# B&R Automation Studio project MVP_ACOPOStrak (part 2)

#### Cyclic.st - Cyclic code
```iecst
PROGRAM _CYCLIC
	CASE Step OF
		CHECK_TRIGGER:
(* When the process is enabled and the assembly is ready,
the process will be activated *)
			IF((CmdEnableProcess) AND (gTrakAsm.Status.Ready))THEN
				MC_BR_TrgPointEnable_AcpTrak_0.Enable := TRUE;
(* If a shuttle passes the triggerpoint then
get the axis reference *)
				IF((MC_BR_TrgPointEnable_AcpTrak_0.Valid) AND
					(MC_BR_TrgPointEnable_AcpTrak_0.EventCount > 0))THEN
					MC_BR_TrgPointGetInfo_AcpTrak_0.Execute := TRUE;
				END_IF
			ELSE (* Else the processpoint will be disabled *)
				MC_BR_TrgPointEnable_AcpTrak_0.Enable := FALSE;
			END_IF
(* If axis reference is available,
save it AND go TO the next step *)
			IF EDGEPOS(MC_BR_TrgPointGetInfo_AcpTrak_0.Done) THEN
(* Save axis reference in local variable for use
in step machine *)
				ShuttleAxis := MC_BR_TrgPointGetInfo_AcpTrak_0.TrgPointInfo.Axis;
				MC_BR_TrgPointGetInfo_AcpTrak_0.Execute := FALSE;
				Step := GET_USERDATA;
				END_IF

		GET_USERDATA:
			(* The userdata is copied on a local variable *)
			MC_BR_ShCopyUserData_AcpTrak_0.Axis := ADR(ShuttleAxis);
			MC_BR_ShCopyUserData_AcpTrak_0.Execute := TRUE;
			MC_BR_ShCopyUserData_AcpTrak_0.DataAddress := ADR(ShuttleUserData);
			MC_BR_ShCopyUserData_AcpTrak_0.DataSize := SIZEOF(ShuttleUserData);
			MC_BR_ShCopyUserData_AcpTrak_0.Mode := mcACPTRAK_USERDATA_GET;
					(* After copying go to the next step *)

			IF EDGEPOS(MC_BR_ShCopyUserData_AcpTrak_0.Done) THEN
				MC_BR_ShCopyUserData_AcpTrak_0.Execute := FALSE;
				Step := PROCESS;
					END_IF

		PROCESS:

			CASE SubStep OF
				0:

					MC_BR_RoutedMoveAbs_AcpTrak_0.Axis := ADR(ShuttleAxis);
					MC_BR_BarrierCommand_AcpTrak_0.Execute := FALSE;

					IF ShuttleUserData.Task = PartsToCell1 OR ShuttleUserData.Task = PartsToCell2 OR ShuttleUserData.Task = MoveAssembly OR ShuttleUserData.Task = MoveSubAssembly THEN
						MC_BR_RoutedMoveAbs_AcpTrak_0.Execute := TRUE;
						MC_BR_RoutedMoveAbs_AcpTrak_0.Sector := ADR(SubSector1_1);
						MC_BR_RoutedMoveAbs_AcpTrak_0.Position := 0.68;
						MC_BR_RoutedMoveAbs_AcpTrak_0.Velocity := 2;
						MC_BR_RoutedMoveAbs_AcpTrak_0.Acceleration := 40;
						MC_BR_RoutedMoveAbs_AcpTrak_0.Deceleration := 40;
						MC_BR_RoutedMoveAbs_AcpTrak_0.Jerk := 0.0;
						MC_BR_RoutedMoveAbs_AcpTrak_0.AdvancedParameters.StartDirection := mcDIR_UNDEFINED;
						MC_BR_RoutedMoveAbs_AcpTrak_0.AdvancedParameters.ShuttleOrientation := mcDIR_POSITIVE;
						MC_BR_RoutedMoveAbs_AcpTrak_0.AdvancedParameters.EndDirection := mcDIR_UNDEFINED;

						IF EDGEPOS (MC_BR_RoutedMoveAbs_AcpTrak_0.Done) THEN
							MC_BR_RoutedMoveAbs_AcpTrak_0.Execute := FALSE;
							SubStep := 10;
						END_IF
					ELSE
						Step := SET_USERDATA;

					END_IF

				10:

					MC_BR_RoutedMoveAbs_AcpTrak_0.Axis := ADR(ShuttleAxis);
					MC_BR_RoutedMoveAbs_AcpTrak_0.Execute := TRUE;

					MC_BR_RoutedMoveAbs_AcpTrak_0.Sector := ADR(SectorTrack6);
					MC_BR_RoutedMoveAbs_AcpTrak_0.Position := 0.1;
					MC_BR_RoutedMoveAbs_AcpTrak_0.Velocity := 2;
					MC_BR_RoutedMoveAbs_AcpTrak_0.Acceleration := 40;
					MC_BR_RoutedMoveAbs_AcpTrak_0.Deceleration := 40;
					MC_BR_RoutedMoveAbs_AcpTrak_0.Jerk := 0.0;
					MC_BR_RoutedMoveAbs_AcpTrak_0.AdvancedParameters.StartDirection := mcDIR_UNDEFINED;
					MC_BR_RoutedMoveAbs_AcpTrak_0.AdvancedParameters.ShuttleOrientation := mcDIR_UNDEFINED;
					MC_BR_RoutedMoveAbs_AcpTrak_0.AdvancedParameters.EndDirection := mcDIR_UNDEFINED;

					IF EDGEPOS (MC_BR_RoutedMoveAbs_AcpTrak_0.Done) THEN
						WaitingLoadOn := TRUE;
					END_IF

					IF LoadOnTrack THEN
						MC_BR_RoutedMoveAbs_AcpTrak_0.Execute := FALSE;
						WaitingLoadOn := FALSE;
						LoadOnTrack := FALSE;
						MC_BR_BarrierCommand_AcpTrak_0.Execute := TRUE;
						MC_BR_BarrierCommand_AcpTrak_0.Command := 1;
						SubStep := 20;
					END_IF

				20:

					MC_BR_BarrierCommand_AcpTrak_0.Execute := FALSE;
					MC_BR_BarrierCommand_AcpTrak_0.Command := 0;
					MC_BR_RoutedMoveAbs_AcpTrak_0.Axis := ADR(ShuttleAxis);
					MC_BR_RoutedMoveAbs_AcpTrak_0.Execute := TRUE;

					MC_BR_RoutedMoveAbs_AcpTrak_0.Sector := ADR(SectorTrack1);
					MC_BR_RoutedMoveAbs_AcpTrak_0.Position := 13;
					MC_BR_RoutedMoveAbs_AcpTrak_0.Velocity := Speed_PP_04;
					MC_BR_RoutedMoveAbs_AcpTrak_0.Acceleration := 20;
					MC_BR_RoutedMoveAbs_AcpTrak_0.Deceleration := 20;
					MC_BR_RoutedMoveAbs_AcpTrak_0.Jerk := 0.0;
					MC_BR_RoutedMoveAbs_AcpTrak_0.AdvancedParameters.StartDirection := mcDIR_UNDEFINED;
					MC_BR_RoutedMoveAbs_AcpTrak_0.AdvancedParameters.ShuttleOrientation := mcDIR_POSITIVE;
					MC_BR_RoutedMoveAbs_AcpTrak_0.AdvancedParameters.EndDirection := mcDIR_UNDEFINED;

					IF EDGEPOS (MC_BR_RoutedMoveAbs_AcpTrak_0.Active) THEN
						MC_BR_RoutedMoveAbs_AcpTrak_0.Execute := FALSE;
						TON_0.IN := TRUE;
						TON_0.PT := T#2s;
						SubStep := 0;
						Step := SET_USERDATA;
					END_IF

			END_CASE

		SET_USERDATA:
			(* The modified userdata will be copied back on the shuttle *)
			MC_BR_ShCopyUserData_AcpTrak_0.Axis := ADR(ShuttleAxis);
			MC_BR_ShCopyUserData_AcpTrak_0.Execute := TRUE;
			MC_BR_ShCopyUserData_AcpTrak_0.DataAddress := ADR(ShuttleUserData);
			MC_BR_ShCopyUserData_AcpTrak_0.DataSize := SIZEOF(ShuttleUserData);
			MC_BR_ShCopyUserData_AcpTrak_0.Mode := mcACPTRAK_USERDATA_SET;

			(* After copying go to the first step and wait for new event *)
			IF EDGEPOS(MC_BR_ShCopyUserData_AcpTrak_0.Done) THEN
				MC_BR_ShCopyUserData_AcpTrak_0.Execute := FALSE;
				Step := CHECK_TRIGGER;
			END_IF
	END_CASE

	IF TON_0.Q THEN
		TON_0.IN := FALSE;
		Track6_Occupied := FALSE;
		MC_BR_BarrierCommand_AcpTrak_0.Execute := TRUE;
	END_IF

	(* Call all function blocks *)
	MC_BR_TrgPointEnable_AcpTrak_0();
	MC_BR_TrgPointGetInfo_AcpTrak_0();
	MC_BR_ShCopyUserData_AcpTrak_0();
	MC_BR_RoutedMoveAbs_AcpTrak_0();
	MC_BR_BarrierCommand_AcpTrak_0();
	TON_0();

END_PROGRAM
PROGRAM _EXIT
END_PROGRAM
```

#### Init.st - Init code
```iecst
PROGRAM _INIT
(* Local variable to enable/disable the the process *)
	Speed_PP_04 := 2;
	CmdEnableProcess := TRUE;
	(* Processpointreference for Functionblocks *)
	MC_BR_TrgPointEnable_AcpTrak_0.ProcessPoint := ADR(PP1);
	MC_BR_TrgPointGetInfo_AcpTrak_0.ProcessPoint := ADR(PP1);
END_PROGRAM
```

#### Types.typ - Local data types
```iecst
TYPE
	Step_enum :
		(
		CHECK_TRIGGER,
		GET_USERDATA,
		PROCESS,
		SET_USERDATA
	);
END_TYPE
```

#### Variables.var - Local variables
```iecst
VAR
	Speed_PP_04 : {REDUND_UNREPLICABLE} REAL := 0.0;
	MC_BR_BarrierCommand_AcpTrak_0 : MC_BR_BarrierCommand_AcpTrak;
	Step : Step_enum;
	MC_BR_TrgPointEnable_AcpTrak_0 : MC_BR_TrgPointEnable_AcpTrak;
	CmdEnableProcess : BOOL;
	MC_BR_TrgPointGetInfo_AcpTrak_0 : MC_BR_TrgPointGetInfo_AcpTrak;
	ShuttleAxis : McAxisType;
	MC_BR_ShCopyUserData_AcpTrak_0 : MC_BR_ShCopyUserData_AcpTrak;
	MC_BR_RoutedMoveAbs_AcpTrak_0 : MC_BR_RoutedMoveAbs_AcpTrak;
	SubStep : UDINT;
	TaskReady : BOOL;
	TON_0 : TON;
	ShuttleUserData : ShuttleUserData_typ;
	MC_BR_RoutedMoveVel_AcpTrak_0 : MC_BR_RoutedMoveVel_AcpTrak;
END_VAR
```

### Program Logical/PP2 (IEC)

#### Variables.var
```iecst
VAR
	Speed_PP_04 : {REDUND_UNREPLICABLE} REAL := 0.0;
	MC_BR_BarrierCommand_AcpTrak_0 : MC_BR_BarrierCommand_AcpTrak;
	Step : Step_enum;
	MC_BR_TrgPointEnable_AcpTrak_0 : MC_BR_TrgPointEnable_AcpTrak;
	CmdEnableProcess : BOOL;
	MC_BR_TrgPointGetInfo_AcpTrak_0 : MC_BR_TrgPointGetInfo_AcpTrak;
	ShuttleAxis : McAxisType;
	MC_BR_ShCopyUserData_AcpTrak_0 : MC_BR_ShCopyUserData_AcpTrak;
	MC_BR_RoutedMoveVel_AcpTrak_0 : MC_BR_RoutedMoveVel_AcpTrak;
	SubStep : UDINT;
	TaskReady : BOOL;
	TaskCompleteCell1 : BOOL;
	ShuttleUserData : ShuttleUserData_typ;
END_VAR
```

#### Cyclic.st
```iecst
PROGRAM _CYCLIC
	CASE Step OF
		CHECK_TRIGGER:
(* When the process is enabled and the assembly is ready,
the process will be activated *)
			IF((CmdEnableProcess) AND (gTrakAsm.Status.Ready))THEN
				MC_BR_TrgPointEnable_AcpTrak_0.Enable := TRUE;
(* If a shuttle passes the triggerpoint then
get the axis reference *)
				IF((MC_BR_TrgPointEnable_AcpTrak_0.Valid) AND
					(MC_BR_TrgPointEnable_AcpTrak_0.EventCount > 0))THEN
					MC_BR_TrgPointGetInfo_AcpTrak_0.Execute := TRUE;
				END_IF
			ELSE (* Else the processpoint will be disabled *)
				MC_BR_TrgPointEnable_AcpTrak_0.Enable := FALSE;
			END_IF
(* If axis reference is available,
save it AND go TO the next step *)
			IF EDGEPOS(MC_BR_TrgPointGetInfo_AcpTrak_0.Done) THEN
(* Save axis reference in local variable for use
in step machine *)
				ShuttleAxis := MC_BR_TrgPointGetInfo_AcpTrak_0.TrgPointInfo.Axis;
				MC_BR_TrgPointGetInfo_AcpTrak_0.Execute := FALSE;
				Step := GET_USERDATA;
				END_IF

		GET_USERDATA:
			(* The userdata is copied on a local variable *)
			MC_BR_ShCopyUserData_AcpTrak_0.Axis := ADR(ShuttleAxis);
			MC_BR_ShCopyUserData_AcpTrak_0.Execute := TRUE;
			MC_BR_ShCopyUserData_AcpTrak_0.DataAddress := ADR(ShuttleUserData);
			MC_BR_ShCopyUserData_AcpTrak_0.DataSize := SIZEOF(ShuttleUserData);
			MC_BR_ShCopyUserData_AcpTrak_0.Mode := mcACPTRAK_USERDATA_GET;
					(* After copying go to the next step *)

			IF EDGEPOS(MC_BR_ShCopyUserData_AcpTrak_0.Done) THEN
				MC_BR_ShCopyUserData_AcpTrak_0.Execute := FALSE;
				Step := PROCESS;
					END_IF

		PROCESS:

		IF ShuttleUserData.Task = PartsToCell1 OR ShuttleUserData.Task = PartsFromCell1 OR ShuttleUserData.Task = MoveAssembly THEN

			MC_BR_RoutedMoveVel_AcpTrak_0.Axis := ADR(ShuttleAxis);
			MC_BR_RoutedMoveVel_AcpTrak_0.Execute := TRUE;
			MC_BR_RoutedMoveVel_AcpTrak_0.Sector := ADR(SectorTrack2);
			MC_BR_RoutedMoveVel_AcpTrak_0.Position := 0;
			MC_BR_RoutedMoveVel_AcpTrak_0.Velocity := Speed_PP_04;
			MC_BR_RoutedMoveVel_AcpTrak_0.RouteVelocity := Speed_PP_04;
			MC_BR_RoutedMoveVel_AcpTrak_0.Acceleration := 10;
			MC_BR_RoutedMoveVel_AcpTrak_0.Deceleration := 10;
			MC_BR_RoutedMoveVel_AcpTrak_0.Jerk := 0.0;
			MC_BR_RoutedMoveVel_AcpTrak_0.AdvancedParameters.StartDirection := mcDIR_UNDEFINED;
			MC_BR_RoutedMoveVel_AcpTrak_0.AdvancedParameters.ShuttleOrientation := mcDIR_NEGATIVE;
			MC_BR_RoutedMoveVel_AcpTrak_0.AdvancedParameters.EndDirection := mcDIR_UNDEFINED;

			IF EDGEPOS (MC_BR_RoutedMoveVel_AcpTrak_0.Active) THEN
				MC_BR_RoutedMoveVel_AcpTrak_0.Execute := FALSE;
				Step := SET_USERDATA;
				END_IF
			ELSE

				MC_BR_RoutedMoveVel_AcpTrak_0.Axis := ADR(ShuttleAxis);
				MC_BR_RoutedMoveVel_AcpTrak_0.Execute := TRUE;
				MC_BR_RoutedMoveVel_AcpTrak_0.Sector := ADR(SectorTrack1);
				MC_BR_RoutedMoveVel_AcpTrak_0.Position := 5;
				MC_BR_RoutedMoveVel_AcpTrak_0.Velocity := Speed_PP_04;
				MC_BR_RoutedMoveVel_AcpTrak_0.RouteVelocity := Speed_PP_04;
				MC_BR_RoutedMoveVel_AcpTrak_0.Acceleration := 10;
				MC_BR_RoutedMoveVel_AcpTrak_0.Deceleration := 10;
				MC_BR_RoutedMoveVel_AcpTrak_0.Jerk := 0.0;
				MC_BR_RoutedMoveVel_AcpTrak_0.AdvancedParameters.StartDirection := mcDIR_POSITIVE;
				MC_BR_RoutedMoveVel_AcpTrak_0.AdvancedParameters.ShuttleOrientation := mcDIR_UNDEFINED;
				MC_BR_RoutedMoveVel_AcpTrak_0.AdvancedParameters.EndDirection := mcDIR_UNDEFINED;

				IF EDGEPOS (MC_BR_RoutedMoveVel_AcpTrak_0.Active) THEN
					MC_BR_RoutedMoveVel_AcpTrak_0.Execute := FALSE;
					Step := SET_USERDATA;
				END_IF
		END_IF

		SET_USERDATA:
			(* The modified userdata will be copied back on the shuttle *)
			MC_BR_ShCopyUserData_AcpTrak_0.Axis := ADR(ShuttleAxis);
			MC_BR_ShCopyUserData_AcpTrak_0.Execute := TRUE;
			MC_BR_ShCopyUserData_AcpTrak_0.DataAddress := ADR(ShuttleUserData);
			MC_BR_ShCopyUserData_AcpTrak_0.DataSize := SIZEOF(ShuttleUserData);
			MC_BR_ShCopyUserData_AcpTrak_0.Mode := mcACPTRAK_USERDATA_SET;

			(* After copying go to the first step and wait for new event *)
			IF EDGEPOS(MC_BR_ShCopyUserData_AcpTrak_0.Done) THEN
				MC_BR_ShCopyUserData_AcpTrak_0.Execute := FALSE;
				Step := CHECK_TRIGGER;
			END_IF
	END_CASE

	(* Call all function blocks *)
	MC_BR_TrgPointEnable_AcpTrak_0();
	MC_BR_TrgPointGetInfo_AcpTrak_0();
	MC_BR_ShCopyUserData_AcpTrak_0();
	MC_BR_RoutedMoveVel_AcpTrak_0();
	MC_BR_BarrierCommand_AcpTrak_0();

END_PROGRAM
PROGRAM _EXIT
END_PROGRAM
```

#### Init.st
```iecst
PROGRAM _INIT
(* Local variable to enable/disable the the process *)
	Speed_PP_04 := 2;
	CmdEnableProcess := TRUE;
	(* Processpointreference for Functionblocks *)
	MC_BR_TrgPointEnable_AcpTrak_0.ProcessPoint := ADR(PP2);
	MC_BR_TrgPointGetInfo_AcpTrak_0.ProcessPoint := ADR(PP2);
END_PROGRAM
```

### Program Logical/PB2 (IEC)

#### Variables.var
```iecst
VAR
	Speed_PP_04 : {REDUND_UNREPLICABLE} REAL := 0.0;
	MC_BR_BarrierCommand_AcpTrak_0 : MC_BR_BarrierCommand_AcpTrak;
	Step : Step_enum;
	MC_BR_TrgPointEnable_AcpTrak_0 : MC_BR_TrgPointEnable_AcpTrak;
	CmdEnableProcess : BOOL;
	MC_BR_TrgPointGetInfo_AcpTrak_0 : MC_BR_TrgPointGetInfo_AcpTrak;
	ShuttleAxis : McAxisType;
	MC_BR_ShCopyUserData_AcpTrak_0 : MC_BR_ShCopyUserData_AcpTrak;
	MC_BR_RoutedMoveAbs_AcpTrak_0 : MC_BR_RoutedMoveAbs_AcpTrak;
	SubStep : UDINT;
	TaskReady : BOOL;
	MC_BR_RoutedMoveVel_AcpTrak_0 : MC_BR_RoutedMoveVel_AcpTrak;
	ShuttleUserData : ShuttleUserData_typ;
END_VAR
```

#### Cyclic.st
```iecst
PROGRAM _CYCLIC
	CASE Step OF
		CHECK_TRIGGER:
(* When the process is enabled and the assembly is ready,
the process will be activated *)
			IF((CmdEnableProcess) AND (gTrakAsm.Status.Ready))THEN
				MC_BR_TrgPointEnable_AcpTrak_0.Enable := TRUE;
(* If a shuttle passes the triggerpoint then
get the axis reference *)
				IF((MC_BR_TrgPointEnable_AcpTrak_0.Valid) AND
					(MC_BR_TrgPointEnable_AcpTrak_0.EventCount > 0))THEN
					MC_BR_TrgPointGetInfo_AcpTrak_0.Execute := TRUE;
				END_IF
			ELSE (* Else the processpoint will be disabled *)
				MC_BR_TrgPointEnable_AcpTrak_0.Enable := FALSE;
			END_IF
(* If axis reference is available,
save it AND go TO the next step *)
			IF EDGEPOS(MC_BR_TrgPointGetInfo_AcpTrak_0.Done) THEN
(* Save axis reference in local variable for use
in step machine *)
				ShuttleAxis := MC_BR_TrgPointGetInfo_AcpTrak_0.TrgPointInfo.Axis;
				MC_BR_TrgPointGetInfo_AcpTrak_0.Execute := FALSE;
				Step := GET_USERDATA;
				END_IF

		GET_USERDATA:
			(* The userdata is copied on a local variable *)
			MC_BR_ShCopyUserData_AcpTrak_0.Axis := ADR(ShuttleAxis);
			MC_BR_ShCopyUserData_AcpTrak_0.Execute := TRUE;
			MC_BR_ShCopyUserData_AcpTrak_0.DataAddress := ADR(ShuttleUserData);
			MC_BR_ShCopyUserData_AcpTrak_0.DataSize := SIZEOF(ShuttleUserData);
			MC_BR_ShCopyUserData_AcpTrak_0.Mode := mcACPTRAK_USERDATA_GET;
					(* After copying go to the next step *)

			IF EDGEPOS(MC_BR_ShCopyUserData_AcpTrak_0.Done) THEN
				MC_BR_ShCopyUserData_AcpTrak_0.Execute := FALSE;
				Step := PROCESS;
					END_IF

		PROCESS:

			CASE SubStep OF
				0:

				MC_BR_RoutedMoveAbs_AcpTrak_0.Axis := ADR(ShuttleAxis);
				MC_BR_RoutedMoveAbs_AcpTrak_0.Execute := TRUE;
				MC_BR_BarrierCommand_AcpTrak_0.Execute := TRUE;
				MC_BR_BarrierCommand_AcpTrak_0.Command := 1;

				MC_BR_RoutedMoveAbs_AcpTrak_0.Sector := ADR(SubSector2_1);
				MC_BR_RoutedMoveAbs_AcpTrak_0.Position := 0.6;
				MC_BR_RoutedMoveAbs_AcpTrak_0.Velocity := Speed_PP_04;

				MC_BR_RoutedMoveAbs_AcpTrak_0.Acceleration := 10;
				MC_BR_RoutedMoveAbs_AcpTrak_0.Deceleration := 10;
				MC_BR_RoutedMoveAbs_AcpTrak_0.Jerk := 0.0;
				MC_BR_RoutedMoveAbs_AcpTrak_0.AdvancedParameters.StartDirection := mcDIR_UNDEFINED;
				MC_BR_RoutedMoveAbs_AcpTrak_0.AdvancedParameters.ShuttleOrientation := mcDIR_NEGATIVE;
				MC_BR_RoutedMoveAbs_AcpTrak_0.AdvancedParameters.EndDirection := mcDIR_UNDEFINED;

				IF EDGEPOS (MC_BR_RoutedMoveAbs_AcpTrak_0.Done) THEN
					MC_BR_RoutedMoveAbs_AcpTrak_0.Execute := FALSE;
					MC_BR_BarrierCommand_AcpTrak_0.Command := 0;
					MC_BR_BarrierCommand_AcpTrak_0.Execute := FALSE;
					WaitingCell1 := TRUE;
					SubStep := 10;

				END_IF

		10:

			IF TaskCompleteCell1 THEN
				MC_BR_RoutedMoveVel_AcpTrak_0.Axis := ADR(ShuttleAxis);
				MC_BR_RoutedMoveVel_AcpTrak_0.Execute := TRUE;
				MC_BR_BarrierCommand_AcpTrak_0.Execute := TRUE;
				MC_BR_RoutedMoveVel_AcpTrak_0.Sector := ADR(SectorTrack1);
				MC_BR_RoutedMoveVel_AcpTrak_0.Position := 4;
				MC_BR_RoutedMoveVel_AcpTrak_0.Velocity := Speed_PP_04;
				MC_BR_RoutedMoveVel_AcpTrak_0.RouteVelocity := Speed_PP_04;
				MC_BR_RoutedMoveVel_AcpTrak_0.Acceleration := 10;
				MC_BR_RoutedMoveVel_AcpTrak_0.Deceleration := 10;
				MC_BR_RoutedMoveVel_AcpTrak_0.Jerk := 0.0;
				MC_BR_RoutedMoveVel_AcpTrak_0.AdvancedParameters.StartDirection := mcDIR_UNDEFINED;
				MC_BR_RoutedMoveVel_AcpTrak_0.AdvancedParameters.ShuttleOrientation := mcDIR_POSITIVE;
				MC_BR_RoutedMoveVel_AcpTrak_0.AdvancedParameters.EndDirection := mcDIR_POSITIVE;

				IF EDGEPOS (MC_BR_RoutedMoveVel_AcpTrak_0.Active) THEN
					MC_BR_RoutedMoveVel_AcpTrak_0.Execute := FALSE;
					MC_BR_BarrierCommand_AcpTrak_0.Execute := FALSE;
					WaitingCell1 := FALSE;
					TaskCompleteCell1 := FALSE;
					SubStep := 0;
					Step := SET_USERDATA;
				END_IF
			END_IF
	END_CASE

		SET_USERDATA:
			(* The modified userdata will be copied back on the shuttle *)
			MC_BR_ShCopyUserData_AcpTrak_0.Axis := ADR(ShuttleAxis);
			MC_BR_ShCopyUserData_AcpTrak_0.Execute := TRUE;
			MC_BR_ShCopyUserData_AcpTrak_0.DataAddress := ADR(ShuttleUserData);
			MC_BR_ShCopyUserData_AcpTrak_0.DataSize := SIZEOF(ShuttleUserData);
			MC_BR_ShCopyUserData_AcpTrak_0.Mode := mcACPTRAK_USERDATA_SET;

			(* After copying go to the first step and wait for new event *)
			IF EDGEPOS(MC_BR_ShCopyUserData_AcpTrak_0.Done) THEN
				MC_BR_ShCopyUserData_AcpTrak_0.Execute := FALSE;
				Step := CHECK_TRIGGER;
			END_IF
	END_CASE

	(* Call all function blocks *)
	MC_BR_TrgPointEnable_AcpTrak_0();
	MC_BR_TrgPointGetInfo_AcpTrak_0();
	MC_BR_ShCopyUserData_AcpTrak_0();
	MC_BR_RoutedMoveAbs_AcpTrak_0();
	MC_BR_BarrierCommand_AcpTrak_0();
	MC_BR_RoutedMoveVel_AcpTrak_0();

END_PROGRAM
PROGRAM _EXIT
END_PROGRAM
```

#### Init.st
```iecst
PROGRAM _INIT
(* Local variable to enable/disable the the process *)
	Speed_PP_04 := 2;
	CmdEnableProcess := TRUE;
	(* Processpointreference for Functionblocks *)
	MC_BR_TrgPointEnable_AcpTrak_0.ProcessPoint := ADR(PB2);
	MC_BR_TrgPointGetInfo_AcpTrak_0.ProcessPoint := ADR(PB2);
	MC_BR_BarrierCommand_AcpTrak_0.ProcessPoint := ADR(PB2);
	MC_BR_BarrierCommand_AcpTrak_0.Command := 1;
END_PROGRAM
```

### Program Logical/PP3 (IEC)

#### Variables.var
```iecst
VAR
	Speed_PP_04 : {REDUND_UNREPLICABLE} REAL := 0.0;
	MC_BR_BarrierCommand_AcpTrak_0 : MC_BR_BarrierCommand_AcpTrak;
	Step : Step_enum;
	MC_BR_TrgPointEnable_AcpTrak_0 : MC_BR_TrgPointEnable_AcpTrak;
	CmdEnableProcess : BOOL;
	MC_BR_TrgPointGetInfo_AcpTrak_0 : MC_BR_TrgPointGetInfo_AcpTrak;
	ShuttleAxis : McAxisType;
	MC_BR_ShCopyUserData_AcpTrak_0 : MC_BR_ShCopyUserData_AcpTrak;
	MC_BR_RoutedMoveVel_AcpTrak_0 : MC_BR_RoutedMoveVel_AcpTrak;
	SubStep : UDINT;
	TaskReady : BOOL;
	TaskCompleteCell2 : BOOL;
	ShuttleUserData : ShuttleUserData_typ;
END_VAR
```

#### Cyclic.st
```iecst
PROGRAM _CYCLIC
	CASE Step OF
		CHECK_TRIGGER:
(* When the process is enabled and the assembly is ready,
the process will be activated *)
			IF((CmdEnableProcess) AND (gTrakAsm.Status.Ready))THEN
				MC_BR_TrgPointEnable_AcpTrak_0.Enable := TRUE;
(* If a shuttle passes the triggerpoint then
get the axis reference *)
				IF((MC_BR_TrgPointEnable_AcpTrak_0.Valid) AND
					(MC_BR_TrgPointEnable_AcpTrak_0.EventCount > 0))THEN
					MC_BR_TrgPointGetInfo_AcpTrak_0.Execute := TRUE;
				END_IF
			ELSE (* Else the processpoint will be disabled *)
				MC_BR_TrgPointEnable_AcpTrak_0.Enable := FALSE;
			END_IF
(* If axis reference is available,
save it AND go TO the next step *)
			IF EDGEPOS(MC_BR_TrgPointGetInfo_AcpTrak_0.Done) THEN
(* Save axis reference in local variable for use
in step machine *)
				ShuttleAxis := MC_BR_TrgPointGetInfo_AcpTrak_0.TrgPointInfo.Axis;
				MC_BR_TrgPointGetInfo_AcpTrak_0.Execute := FALSE;
				Step := GET_USERDATA;
				END_IF

		GET_USERDATA:
			(* The userdata is copied on a local variable *)
			MC_BR_ShCopyUserData_AcpTrak_0.Axis := ADR(ShuttleAxis);
			MC_BR_ShCopyUserData_AcpTrak_0.Execute := TRUE;
			MC_BR_ShCopyUserData_AcpTrak_0.DataAddress := ADR(ShuttleUserData);
			MC_BR_ShCopyUserData_AcpTrak_0.DataSize := SIZEOF(ShuttleUserData);
			MC_BR_ShCopyUserData_AcpTrak_0.Mode := mcACPTRAK_USERDATA_GET;
					(* After copying go to the next step *)

			IF EDGEPOS(MC_BR_ShCopyUserData_AcpTrak_0.Done) THEN
				MC_BR_ShCopyUserData_AcpTrak_0.Execute := FALSE;
				Step := PROCESS;
					END_IF

		PROCESS:

		IF ShuttleUserData.Task = PartsToCell2 OR ShuttleUserData.Task = PartsFromCell2 OR ShuttleUserData.Task = MoveAssembly OR ShuttleUserData.Task = MoveSubAssembly THEN

			MC_BR_RoutedMoveVel_AcpTrak_0.Axis := ADR(ShuttleAxis);
			MC_BR_RoutedMoveVel_AcpTrak_0.Execute := TRUE;
			MC_BR_RoutedMoveVel_AcpTrak_0.Sector := ADR(SubSector3_1);
			MC_BR_RoutedMoveVel_AcpTrak_0.Position := 0;
			MC_BR_RoutedMoveVel_AcpTrak_0.Velocity := Speed_PP_04;
			MC_BR_RoutedMoveVel_AcpTrak_0.RouteVelocity := Speed_PP_04;
			MC_BR_RoutedMoveVel_AcpTrak_0.Acceleration := 10;
			MC_BR_RoutedMoveVel_AcpTrak_0.Deceleration := 10;
			MC_BR_RoutedMoveVel_AcpTrak_0.Jerk := 0.0;
			MC_BR_RoutedMoveVel_AcpTrak_0.AdvancedParameters.StartDirection := mcDIR_UNDEFINED;
			MC_BR_RoutedMoveVel_AcpTrak_0.AdvancedParameters.ShuttleOrientation := mcDIR_NEGATIVE;
			MC_BR_RoutedMoveVel_AcpTrak_0.AdvancedParameters.EndDirection := mcDIR_UNDEFINED;

			IF EDGEPOS (MC_BR_RoutedMoveVel_AcpTrak_0.Active) THEN
				MC_BR_RoutedMoveVel_AcpTrak_0.Execute := FALSE;
				Step := SET_USERDATA;
				END_IF
			ELSE
				Step := SET_USERDATA;
		END_IF

		SET_USERDATA:
			(* The modified userdata will be copied back on the shuttle *)
			MC_BR_ShCopyUserData_AcpTrak_0.Axis := ADR(ShuttleAxis);
			MC_BR_ShCopyUserData_AcpTrak_0.Execute := TRUE;
			MC_BR_ShCopyUserData_AcpTrak_0.DataAddress := ADR(ShuttleUserData);
			MC_BR_ShCopyUserData_AcpTrak_0.DataSize := SIZEOF(ShuttleUserData);
			MC_BR_ShCopyUserData_AcpTrak_0.Mode := mcACPTRAK_USERDATA_SET;

			(* After copying go to the first step and wait for new event *)
			IF EDGEPOS(MC_BR_ShCopyUserData_AcpTrak_0.Done) THEN
				MC_BR_ShCopyUserData_AcpTrak_0.Execute := FALSE;
				Step := CHECK_TRIGGER;
			END_IF
	END_CASE

	(* Call all function blocks *)
	MC_BR_TrgPointEnable_AcpTrak_0();
	MC_BR_TrgPointGetInfo_AcpTrak_0();
	MC_BR_ShCopyUserData_AcpTrak_0();
	MC_BR_RoutedMoveVel_AcpTrak_0();
	MC_BR_BarrierCommand_AcpTrak_0();

END_PROGRAM
PROGRAM _EXIT
END_PROGRAM
```

#### Init.st
```iecst
PROGRAM _INIT
(* Local variable to enable/disable the the process *)
	Speed_PP_04 := 2;
	CmdEnableProcess := TRUE;
	(* Processpointreference for Functionblocks *)
	MC_BR_TrgPointEnable_AcpTrak_0.ProcessPoint := ADR(PP3);
	MC_BR_TrgPointGetInfo_AcpTrak_0.ProcessPoint := ADR(PP3);
END_PROGRAM
```

### Program Logical/PB3 (IEC)

#### Variables.var
```iecst
VAR
	MC_BR_RoutedMoveVel_AcpTrak_0 : MC_BR_RoutedMoveVel_AcpTrak;
	Speed_PP_04 : {REDUND_UNREPLICABLE} REAL := 0.0;
	MC_BR_BarrierCommand_AcpTrak_0 : MC_BR_BarrierCommand_AcpTrak;
	Step : Step_enum;
	MC_BR_TrgPointEnable_AcpTrak_0 : MC_BR_TrgPointEnable_AcpTrak;
	CmdEnableProcess : BOOL;
	MC_BR_TrgPointGetInfo_AcpTrak_0 : MC_BR_TrgPointGetInfo_AcpTrak;
	ShuttleAxis : McAxisType;
	MC_BR_ShCopyUserData_AcpTrak_0 : MC_BR_ShCopyUserData_AcpTrak;
	MC_BR_RoutedMoveAbs_AcpTrak_0 : MC_BR_RoutedMoveAbs_AcpTrak;
	SubStep : UDINT;
	TaskReady : BOOL;
	ShuttleUserData : ShuttleUserData_typ;
END_VAR
```

#### Cyclic.st
```iecst
PROGRAM _CYCLIC
	CASE Step OF
		CHECK_TRIGGER:
(* When the process is enabled and the assembly is ready,
the process will be activated *)
			IF((CmdEnableProcess) AND (gTrakAsm.Status.Ready))THEN
				MC_BR_TrgPointEnable_AcpTrak_0.Enable := TRUE;
(* If a shuttle passes the triggerpoint then
get the axis reference *)
				IF((MC_BR_TrgPointEnable_AcpTrak_0.Valid) AND
					(MC_BR_TrgPointEnable_AcpTrak_0.EventCount > 0))THEN
					MC_BR_TrgPointGetInfo_AcpTrak_0.Execute := TRUE;
				END_IF
			ELSE (* Else the processpoint will be disabled *)
				MC_BR_TrgPointEnable_AcpTrak_0.Enable := FALSE;
			END_IF
(* If axis reference is available,
save it AND go TO the next step *)
			IF EDGEPOS(MC_BR_TrgPointGetInfo_AcpTrak_0.Done) THEN
(* Save axis reference in local variable for use
in step machine *)
				ShuttleAxis := MC_BR_TrgPointGetInfo_AcpTrak_0.TrgPointInfo.Axis;
				MC_BR_TrgPointGetInfo_AcpTrak_0.Execute := FALSE;
				Step := GET_USERDATA;
				END_IF

		GET_USERDATA:
			(* The userdata is copied on a local variable *)
			MC_BR_ShCopyUserData_AcpTrak_0.Axis := ADR(ShuttleAxis);
			MC_BR_ShCopyUserData_AcpTrak_0.Execute := TRUE;
			MC_BR_ShCopyUserData_AcpTrak_0.DataAddress := ADR(ShuttleUserData);
			MC_BR_ShCopyUserData_AcpTrak_0.DataSize := SIZEOF(ShuttleUserData);
			MC_BR_ShCopyUserData_AcpTrak_0.Mode := mcACPTRAK_USERDATA_GET;
					(* After copying go to the next step *)

			IF EDGEPOS(MC_BR_ShCopyUserData_AcpTrak_0.Done) THEN
				MC_BR_ShCopyUserData_AcpTrak_0.Execute := FALSE;
				Step := PROCESS;
					END_IF

		PROCESS:

			CASE SubStep OF
				0:

					MC_BR_RoutedMoveAbs_AcpTrak_0.Axis := ADR(ShuttleAxis);
					MC_BR_RoutedMoveAbs_AcpTrak_0.Execute := TRUE;
					MC_BR_BarrierCommand_AcpTrak_0.Execute := TRUE;
					MC_BR_BarrierCommand_AcpTrak_0.Command := 1;
					MC_BR_RoutedMoveAbs_AcpTrak_0.Sector := ADR(SubSector3_1);
					MC_BR_RoutedMoveAbs_AcpTrak_0.Position := 0.6;
					MC_BR_RoutedMoveAbs_AcpTrak_0.Velocity := Speed_PP_04;

					MC_BR_RoutedMoveAbs_AcpTrak_0.Acceleration := 10;
					MC_BR_RoutedMoveAbs_AcpTrak_0.Deceleration := 10;
					MC_BR_RoutedMoveAbs_AcpTrak_0.Jerk := 0.0;
					MC_BR_RoutedMoveAbs_AcpTrak_0.AdvancedParameters.StartDirection := mcDIR_UNDEFINED;
					MC_BR_RoutedMoveAbs_AcpTrak_0.AdvancedParameters.ShuttleOrientation := mcDIR_NEGATIVE;
					MC_BR_RoutedMoveAbs_AcpTrak_0.AdvancedParameters.EndDirection := mcDIR_UNDEFINED;

					IF EDGEPOS (MC_BR_RoutedMoveAbs_AcpTrak_0.Done) THEN
						MC_BR_RoutedMoveAbs_AcpTrak_0.Execute := FALSE;
						MC_BR_BarrierCommand_AcpTrak_0.Command := 0;
						MC_BR_BarrierCommand_AcpTrak_0.Execute := FALSE;
						WaitingCell2 := TRUE;
						SubStep := 10;

					END_IF

				10:

					IF TaskCompleteCell2 THEN
						MC_BR_RoutedMoveVel_AcpTrak_0.Axis := ADR(ShuttleAxis);
						MC_BR_RoutedMoveVel_AcpTrak_0.Execute := TRUE;
						MC_BR_BarrierCommand_AcpTrak_0.Execute := TRUE;
						MC_BR_RoutedMoveVel_AcpTrak_0.Sector := ADR(SectorTrack1);
						MC_BR_RoutedMoveVel_AcpTrak_0.Position := 5;
						MC_BR_RoutedMoveVel_AcpTrak_0.Velocity := Speed_PP_04;
						MC_BR_RoutedMoveVel_AcpTrak_0.RouteVelocity := Speed_PP_04;
						MC_BR_RoutedMoveVel_AcpTrak_0.Acceleration := 10;
						MC_BR_RoutedMoveVel_AcpTrak_0.Deceleration := 10;
						MC_BR_RoutedMoveVel_AcpTrak_0.Jerk := 0.0;
						MC_BR_RoutedMoveVel_AcpTrak_0.AdvancedParameters.StartDirection := mcDIR_UNDEFINED;
						MC_BR_RoutedMoveVel_AcpTrak_0.AdvancedParameters.ShuttleOrientation := mcDIR_POSITIVE;
						MC_BR_RoutedMoveVel_AcpTrak_0.AdvancedParameters.EndDirection := mcDIR_POSITIVE;

						IF EDGEPOS (MC_BR_RoutedMoveVel_AcpTrak_0.Active) THEN
							MC_BR_RoutedMoveVel_AcpTrak_0.Execute := FALSE;
							MC_BR_BarrierCommand_AcpTrak_0.Execute := FALSE;
							WaitingCell2 := FALSE;
							TaskCompleteCell2 := FALSE;
							SubStep := 0;
							Step := SET_USERDATA;
						END_IF
					END_IF
			END_CASE

		SET_USERDATA:
			(* The modified userdata will be copied back on the shuttle *)
			MC_BR_ShCopyUserData_AcpTrak_0.Axis := ADR(ShuttleAxis);
			MC_BR_ShCopyUserData_AcpTrak_0.Execute := TRUE;
			MC_BR_ShCopyUserData_AcpTrak_0.DataAddress := ADR(ShuttleUserData);
			MC_BR_ShCopyUserData_AcpTrak_0.DataSize := SIZEOF(ShuttleUserData);
			MC_BR_ShCopyUserData_AcpTrak_0.Mode := mcACPTRAK_USERDATA_SET;

			(* After copying go to the first step and wait for new event *)
			IF EDGEPOS(MC_BR_ShCopyUserData_AcpTrak_0.Done) THEN
				MC_BR_ShCopyUserData_AcpTrak_0.Execute := FALSE;
				Step := CHECK_TRIGGER;
			END_IF
	END_CASE

	(* Call all function blocks *)
	MC_BR_TrgPointEnable_AcpTrak_0();
	MC_BR_TrgPointGetInfo_AcpTrak_0();
	MC_BR_ShCopyUserData_AcpTrak_0();
	MC_BR_RoutedMoveAbs_AcpTrak_0();
	MC_BR_BarrierCommand_AcpTrak_0();
	MC_BR_RoutedMoveVel_AcpTrak_0();

END_PROGRAM
PROGRAM _EXIT
END_PROGRAM
```

#### Init.st
```iecst
PROGRAM _INIT
(* Local variable to enable/disable the the process *)
	Speed_PP_04 := 2;
	CmdEnableProcess := TRUE;
	(* Processpointreference for Functionblocks *)
	MC_BR_TrgPointEnable_AcpTrak_0.ProcessPoint := ADR(PB3);
	MC_BR_TrgPointGetInfo_AcpTrak_0.ProcessPoint := ADR(PB3);
	MC_BR_BarrierCommand_AcpTrak_0.ProcessPoint := ADR(PB3);
	MC_BR_BarrierCommand_AcpTrak_0.Command := 1;
END_PROGRAM
```

### Program Logical/PP4 (IEC)

#### Variables.var
```iecst
VAR
	Close : BOOL;
	Speed_PP_04 : {REDUND_UNREPLICABLE} REAL := 0.0;
	MC_BR_BarrierCommand_AcpTrak_0 : MC_BR_BarrierCommand_AcpTrak;
	Step : Step_enum;
	MC_BR_TrgPointEnable_AcpTrak_0 : MC_BR_TrgPointEnable_AcpTrak;
	CmdEnableProcess : BOOL;
	MC_BR_TrgPointGetInfo_AcpTrak_0 : MC_BR_TrgPointGetInfo_AcpTrak;
	ShuttleAxis : McAxisType;
	MC_BR_ShCopyUserData_AcpTrak_0 : MC_BR_ShCopyUserData_AcpTrak;
	MC_BR_RoutedMoveAbs_AcpTrak_0 : MC_BR_RoutedMoveAbs_AcpTrak;
	SubStep : UDINT;
	TaskReady : BOOL;
	TON_0 : TON;
	MC_BR_RoutedMoveVel_AcpTrak_0 : MC_BR_RoutedMoveVel_AcpTrak;
	ShuttleUserData : ShuttleUserData_typ;
END_VAR
```

#### Cyclic.st
```iecst
PROGRAM _CYCLIC
	CASE Step OF
		CHECK_TRIGGER:
(* When the process is enabled and the assembly is ready,
the process will be activated *)
			IF((CmdEnableProcess) AND (gTrakAsm.Status.Ready))THEN
				MC_BR_TrgPointEnable_AcpTrak_0.Enable := TRUE;
(* If a shuttle passes the triggerpoint then
get the axis reference *)
				IF((MC_BR_TrgPointEnable_AcpTrak_0.Valid) AND
					(MC_BR_TrgPointEnable_AcpTrak_0.EventCount > 0))THEN
					MC_BR_TrgPointGetInfo_AcpTrak_0.Execute := TRUE;
				END_IF
			ELSE (* Else the processpoint will be disabled *)
				MC_BR_TrgPointEnable_AcpTrak_0.Enable := FALSE;
			END_IF
(* If axis reference is available,
save it AND go TO the next step *)
			IF EDGEPOS(MC_BR_TrgPointGetInfo_AcpTrak_0.Done) THEN
(* Save axis reference in local variable for use
in step machine *)
				ShuttleAxis := MC_BR_TrgPointGetInfo_AcpTrak_0.TrgPointInfo.Axis;
				MC_BR_TrgPointGetInfo_AcpTrak_0.Execute := FALSE;
				Step := GET_USERDATA;
				END_IF

		GET_USERDATA:
			(* The userdata is copied on a local variable *)
			MC_BR_ShCopyUserData_AcpTrak_0.Axis := ADR(ShuttleAxis);
			MC_BR_ShCopyUserData_AcpTrak_0.Execute := TRUE;
			MC_BR_ShCopyUserData_AcpTrak_0.DataAddress := ADR(ShuttleUserData);
			MC_BR_ShCopyUserData_AcpTrak_0.DataSize := SIZEOF(ShuttleUserData);
			MC_BR_ShCopyUserData_AcpTrak_0.Mode := mcACPTRAK_USERDATA_GET;
					(* After copying go to the next step *)

			IF EDGEPOS(MC_BR_ShCopyUserData_AcpTrak_0.Done) THEN
				MC_BR_ShCopyUserData_AcpTrak_0.Execute := FALSE;
				Step := PROCESS;
					END_IF

		PROCESS:

			CASE SubStep OF
				0:

					IF ShuttleUserData.Task = PartsFromCell1 OR ShuttleUserData.Task = PartsFromCell2 OR ShuttleUserData.Task = MoveAssembly THEN

						IF NOT OutletBarrierLocked THEN
							OutletBarrierLocked :=TRUE;
						END_IF
						MC_BR_RoutedMoveAbs_AcpTrak_0.Execute := TRUE;
						MC_BR_RoutedMoveAbs_AcpTrak_0.Axis := ADR(ShuttleAxis);
						MC_BR_RoutedMoveAbs_AcpTrak_0.Sector := ADR(SectorTrack5);
						MC_BR_RoutedMoveAbs_AcpTrak_0.Position := 0.1;
						MC_BR_RoutedMoveAbs_AcpTrak_0.Velocity := 2;
						MC_BR_RoutedMoveAbs_AcpTrak_0.Acceleration := 10;
						MC_BR_RoutedMoveAbs_AcpTrak_0.Deceleration := 10;
						MC_BR_RoutedMoveAbs_AcpTrak_0.Jerk := 0.0;
						MC_BR_RoutedMoveAbs_AcpTrak_0.AdvancedParameters.StartDirection := mcDIR_UNDEFINED;
						MC_BR_RoutedMoveAbs_AcpTrak_0.AdvancedParameters.ShuttleOrientation := mcDIR_NEGATIVE;
						MC_BR_RoutedMoveAbs_AcpTrak_0.AdvancedParameters.EndDirection := mcDIR_UNDEFINED;
						Track5_Occupied := TRUE;

						IF EDGEPOS (MC_BR_RoutedMoveAbs_AcpTrak_0.Done) THEN
						MC_BR_RoutedMoveAbs_AcpTrak_0.Execute := FALSE;
						WaitingLoadOff := TRUE;
						SubStep := 10;
						END_IF
					ELSE
						Step := SET_USERDATA;

					END_IF

				10:

				IF LoadOffTrack THEN

					TON_0.IN := TRUE;
					TON_0.PT := T#2s;

					IF TON_0.Q THEN
					MC_BR_RoutedMoveAbs_AcpTrak_0.Axis := ADR(ShuttleAxis);
					MC_BR_RoutedMoveAbs_AcpTrak_0.Execute := TRUE;
					MC_BR_RoutedMoveAbs_AcpTrak_0.Sector := ADR(SubSector1_4);
					MC_BR_RoutedMoveAbs_AcpTrak_0.Position := 0.6;
					MC_BR_RoutedMoveAbs_AcpTrak_0.Velocity := 2;
					MC_BR_RoutedMoveAbs_AcpTrak_0.Acceleration := 10;
					MC_BR_RoutedMoveAbs_AcpTrak_0.Deceleration := 10;
					MC_BR_RoutedMoveAbs_AcpTrak_0.Jerk := 0.0;
					MC_BR_RoutedMoveAbs_AcpTrak_0.AdvancedParameters.StartDirection := mcDIR_POSITIVE;
					MC_BR_RoutedMoveAbs_AcpTrak_0.AdvancedParameters.ShuttleOrientation := mcDIR_POSITIVE;
					MC_BR_RoutedMoveAbs_AcpTrak_0.AdvancedParameters.EndDirection := mcDIR_NEGATIVE;

					IF EDGEPOS (MC_BR_RoutedMoveAbs_AcpTrak_0.Done) THEN
							MC_BR_RoutedMoveAbs_AcpTrak_0.Execute := FALSE;
							LoadOffTrack := FALSE;
							WaitingLoadOff := FALSE;
							TON_0.IN := FALSE;

							SubStep := 20;
					END_IF
					END_IF
				END_IF

				20:

					MC_BR_RoutedMoveVel_AcpTrak_0.Axis := ADR(ShuttleAxis);
					MC_BR_RoutedMoveVel_AcpTrak_0.Execute := TRUE;
					MC_BR_RoutedMoveVel_AcpTrak_0.Sector := ADR(SectorTrack1);
					MC_BR_RoutedMoveVel_AcpTrak_0.Position := 10;
					MC_BR_RoutedMoveVel_AcpTrak_0.Velocity := Speed_PP_04;
					MC_BR_RoutedMoveVel_AcpTrak_0.RouteVelocity := Speed_PP_04;
					MC_BR_RoutedMoveVel_AcpTrak_0.Acceleration := 10;
					MC_BR_RoutedMoveVel_AcpTrak_0.Deceleration := 10;
					MC_BR_RoutedMoveVel_AcpTrak_0.Jerk := 0.0;
					MC_BR_RoutedMoveVel_AcpTrak_0.AdvancedParameters.StartDirection := mcDIR_POSITIVE;
					MC_BR_RoutedMoveVel_AcpTrak_0.AdvancedParameters.ShuttleOrientation := mcDIR_POSITIVE;
					MC_BR_RoutedMoveVel_AcpTrak_0.AdvancedParameters.EndDirection := mcDIR_UNDEFINED;

					IF EDGEPOS (MC_BR_RoutedMoveVel_AcpTrak_0.Active) THEN
						MC_BR_RoutedMoveVel_AcpTrak_0.Execute := FALSE;
						Track5_Occupied := FALSE;

						IF WaitingBarrier AND Locked THEN
							TriggerCount := TRUE;
							WaitingBarrier := FALSE;
							Locked := FALSE;
						ELSIF WaitingBarrier AND NOT Locked THEN
							TriggerCount := TRUE;
							WaitingBarrier := FALSE;
							OutletBarrierLocked := FALSE;
						ELSE
							OutletBarrierLocked := FALSE;
						END_IF
						SubStep := 0;
						Step := SET_USERDATA;
					END_IF

			END_CASE

		SET_USERDATA:
			(* The modified userdata will be copied back on the shuttle *)
			MC_BR_ShCopyUserData_AcpTrak_0.Axis := ADR(ShuttleAxis);
			MC_BR_ShCopyUserData_AcpTrak_0.Execute := TRUE;
			MC_BR_ShCopyUserData_AcpTrak_0.DataAddress := ADR(ShuttleUserData);
			MC_BR_ShCopyUserData_AcpTrak_0.DataSize := SIZEOF(ShuttleUserData);
			MC_BR_ShCopyUserData_AcpTrak_0.Mode := mcACPTRAK_USERDATA_SET;

			(* After copying go to the first step and wait for new event *)
			IF EDGEPOS(MC_BR_ShCopyUserData_AcpTrak_0.Done) THEN
				MC_BR_ShCopyUserData_AcpTrak_0.Execute := FALSE;
				Step := CHECK_TRIGGER;
			END_IF
	END_CASE

	IF OutletBarrierLocked AND TriggerCount THEN
		MC_BR_BarrierCommand_AcpTrak_0.Command := 2;
		MC_BR_BarrierCommand_AcpTrak_0.Execute := TRUE;
		TriggerCount := FALSE;
	ELSIF NOT OutletBarrierLocked AND TriggerCount THEN
		MC_BR_BarrierCommand_AcpTrak_0.Command := 2;
		MC_BR_BarrierCommand_AcpTrak_0.Execute := TRUE;
		TriggerCount := FALSE;
	ELSE
		MC_BR_BarrierCommand_AcpTrak_0.Execute := FALSE;
	END_IF

	(* Call all function blocks *)
	MC_BR_TrgPointEnable_AcpTrak_0();
	MC_BR_TrgPointGetInfo_AcpTrak_0();
	MC_BR_ShCopyUserData_AcpTrak_0();
	MC_BR_RoutedMoveAbs_AcpTrak_0();
	MC_BR_RoutedMoveVel_AcpTrak_0();
	MC_BR_BarrierCommand_AcpTrak_0();
	TON_0();

END_PROGRAM
PROGRAM _EXIT
END_PROGRAM
```

#### Init.st
```iecst
PROGRAM _INIT
(* Local variable to enable/disable the the process *)
	Speed_PP_04 := 2;
	CmdEnableProcess := TRUE;
	(* Processpointreference for Functionblocks *)
	MC_BR_TrgPointEnable_AcpTrak_0.ProcessPoint := ADR(PP4);
	MC_BR_TrgPointGetInfo_AcpTrak_0.ProcessPoint := ADR(PP4);
	MC_BR_BarrierCommand_AcpTrak_0.ProcessPoint := ADR(PP4);
	MC_BR_BarrierCommand_AcpTrak_0.Command := 1;
	MC_BR_BarrierCommand_AcpTrak_0.Execute := TRUE;
	MC_BR_BarrierCommand_AcpTrak_0.AdvancedParameters.TicketCount := 1;
	MC_BR_BarrierCommand_AcpTrak_0();
END_PROGRAM
```

### Program Logical/PP5 (IEC)

#### Variables.var
```iecst
VAR
	MC_BR_RoutedMoveVel_AcpTrak_0 : MC_BR_RoutedMoveVel_AcpTrak;
	WaitingLoadOff : BOOL;
	Speed_PP_04 : {REDUND_UNREPLICABLE} REAL := 0.0;
	MC_BR_BarrierCommand_AcpTrak_0 : MC_BR_BarrierCommand_AcpTrak;
	Step : Step_enum;
	MC_BR_TrgPointEnable_AcpTrak_0 : MC_BR_TrgPointEnable_AcpTrak;
	CmdEnableProcess : BOOL;
	MC_BR_TrgPointGetInfo_AcpTrak_0 : MC_BR_TrgPointGetInfo_AcpTrak;
	ShuttleAxis : McAxisType;
	MC_BR_ShCopyUserData_AcpTrak_0 : MC_BR_ShCopyUserData_AcpTrak;
	MC_BR_RoutedMoveAbs_AcpTrak_0 : MC_BR_RoutedMoveAbs_AcpTrak;
	SubStep : UDINT;
	TaskReady : BOOL;
	TON_0 : TON;
	ShuttleUserData : ShuttleUserData_typ;
END_VAR
```

#### Cyclic.st
```iecst
PROGRAM _CYCLIC
	CASE Step OF
		CHECK_TRIGGER:
(* When the process is enabled and the assembly is ready,
the process will be activated *)
			IF((CmdEnableProcess) AND (gTrakAsm.Status.Ready))THEN
				MC_BR_TrgPointEnable_AcpTrak_0.Enable := TRUE;
(* If a shuttle passes the triggerpoint then
get the axis reference *)
				IF((MC_BR_TrgPointEnable_AcpTrak_0.Valid) AND
					(MC_BR_TrgPointEnable_AcpTrak_0.EventCount > 0))THEN
					MC_BR_TrgPointGetInfo_AcpTrak_0.Execute := TRUE;
				END_IF
			ELSE (* Else the processpoint will be disabled *)
				MC_BR_TrgPointEnable_AcpTrak_0.Enable := FALSE;
			END_IF
(* If axis reference is available,
save it AND go TO the next step *)
			IF EDGEPOS(MC_BR_TrgPointGetInfo_AcpTrak_0.Done) THEN
(* Save axis reference in local variable for use
in step machine *)
				ShuttleAxis := MC_BR_TrgPointGetInfo_AcpTrak_0.TrgPointInfo.Axis;
				MC_BR_TrgPointGetInfo_AcpTrak_0.Execute := FALSE;
				Step := GET_USERDATA;
				END_IF

		GET_USERDATA:
			(* The userdata is copied on a local variable *)
			MC_BR_ShCopyUserData_AcpTrak_0.Axis := ADR(ShuttleAxis);
			MC_BR_ShCopyUserData_AcpTrak_0.Execute := TRUE;
			MC_BR_ShCopyUserData_AcpTrak_0.DataAddress := ADR(ShuttleUserData);
			MC_BR_ShCopyUserData_AcpTrak_0.DataSize := SIZEOF(ShuttleUserData);
			MC_BR_ShCopyUserData_AcpTrak_0.Mode := mcACPTRAK_USERDATA_GET;
					(* After copying go to the next step *)

			IF EDGEPOS(MC_BR_ShCopyUserData_AcpTrak_0.Done) THEN
				MC_BR_ShCopyUserData_AcpTrak_0.Execute := FALSE;
				Step := PROCESS;
					END_IF

		PROCESS:

			CASE SubStep OF
				0:

					IF (ShuttleUserData.Task = PartsFromCell1 OR ShuttleUserData.Task = PartsFromCell2 OR ShuttleUserData.Task = MoveAssembly) AND NOT Locked AND NOT OutletBarrierLocked THEN
						OutletBarrierLocked := TRUE;
						TriggerCount := TRUE;
						Step := SET_USERDATA;
					ELSIF (ShuttleUserData.Task = PartsToCell1 OR ShuttleUserData.Task = PartsToCell2 OR ShuttleUserData.Task = MoveSubAssembly OR ShuttleUserData.Task = NoTask) AND NOT LoadOffTrack THEN
						TriggerCount := TRUE;
						Step := SET_USERDATA;
					ELSIF LoadOffTrack AND (ShuttleUserData.Task = PartsToCell1 OR ShuttleUserData.Task = PartsToCell2 OR ShuttleUserData.Task = MoveSubAssembly OR ShuttleUserData.Task = NoTask) THEN
						WaitingBarrier := TRUE;
					ELSE
						Locked := TRUE;
						WaitingBarrier := TRUE;
						Step := SET_USERDATA;
					END_IF

				10:

			END_CASE

		SET_USERDATA:
			(* The modified userdata will be copied back on the shuttle *)
			MC_BR_ShCopyUserData_AcpTrak_0.Axis := ADR(ShuttleAxis);
			MC_BR_ShCopyUserData_AcpTrak_0.Execute := TRUE;
			MC_BR_ShCopyUserData_AcpTrak_0.DataAddress := ADR(ShuttleUserData);
			MC_BR_ShCopyUserData_AcpTrak_0.DataSize := SIZEOF(ShuttleUserData);
			MC_BR_ShCopyUserData_AcpTrak_0.Mode := mcACPTRAK_USERDATA_SET;

			(* After copying go to the first step and wait for new event *)
			IF EDGEPOS(MC_BR_ShCopyUserData_AcpTrak_0.Done) THEN
				MC_BR_ShCopyUserData_AcpTrak_0.Execute := FALSE;
				Step := CHECK_TRIGGER;
			END_IF
	END_CASE

	(* Call all function blocks *)
	MC_BR_TrgPointEnable_AcpTrak_0();
	MC_BR_TrgPointGetInfo_AcpTrak_0();
	MC_BR_ShCopyUserData_AcpTrak_0();
	MC_BR_RoutedMoveAbs_AcpTrak_0();
	MC_BR_RoutedMoveVel_AcpTrak_0();
	TON_0();

END_PROGRAM
PROGRAM _EXIT
END_PROGRAM
```

#### Init.st
```iecst
PROGRAM _INIT
(* Local variable to enable/disable the the process *)
	Speed_PP_04 := 2;
	CmdEnableProcess := TRUE;
	(* Processpointreference for Functionblocks *)
	MC_BR_TrgPointEnable_AcpTrak_0.ProcessPoint := ADR(PP5);
	MC_BR_TrgPointGetInfo_AcpTrak_0.ProcessPoint := ADR(PP5);
END_PROGRAM
```
